TEXTLIST TL_E_INSTANCE
  1 = 'BUFFER_INFEED'
  2 = 'INFEED'
  3 = 'BUFFER_OUTFEED_ROBOT'
  4 = 'OUTFEED_ROBOT_R1'
  5 = 'OUTFEED_ROBOT_R2'
  6 = 'SENDER_FAST'
  7 = 'SENDER_BUFFER_INFEED'
   = ''
END_TEXTLIST

(* stored: Version 1.1.0.1, ProductVersion 3.1.4024.15
   TextList TL_E_INSTANCE: Id {4e59c0b3-ad4c-49a5-8bf8-ec730d21fbcf} *)
